// TIA Portal V18 export
FUNCTION_BLOCK "Control_Buttons_Manipulate"   // FB24, LAD
{ S7_Optimized_Access := 'TRUE' }
VERSION : 0.1
// Simple control block to activate printhead motion in X and Y direction
// stored: AutoNumber true, IsIECCheckEnabled false, IsRetainMemResEnabled false, MemoryReserve 100, SetENOAutomatically false, UDAEnableTagReadback false
   VAR_INPUT
      JogInZ1pos : Bool;
      JogInZ1neg : Bool;
      JogInZ2pos : Bool;
      JogInZ2neg : Bool;
      InXhome : Bool;
      InYhome : Bool;
      InZ1home : Bool;
      InZ2home : Bool;
      MovePermission : Bool;
      ReadyDevices : Bool;
   END_VAR
   VAR_OUTPUT
      JogOutXpos : Bool;
      JogOutXneg : Bool;
      JogOutYpos : Bool;
      JogOutYneg : Bool;
      JogOutZ1pos : Bool;
      JogOutZ1neg : Bool;
      JogOutZ2pos : Bool;
      JogOutZ2neg : Bool;
      XHoming : Bool;
      YHoming : Bool;
      Z1Homing : Bool;
      Z2Homing : Bool;
      StartMachine : Bool;
   END_VAR
   VAR
      ButtonsReadyToRead : Bool;
      XYmoveout : Bool;
   END_VAR
BEGIN

REGION Network 1: Start Machine
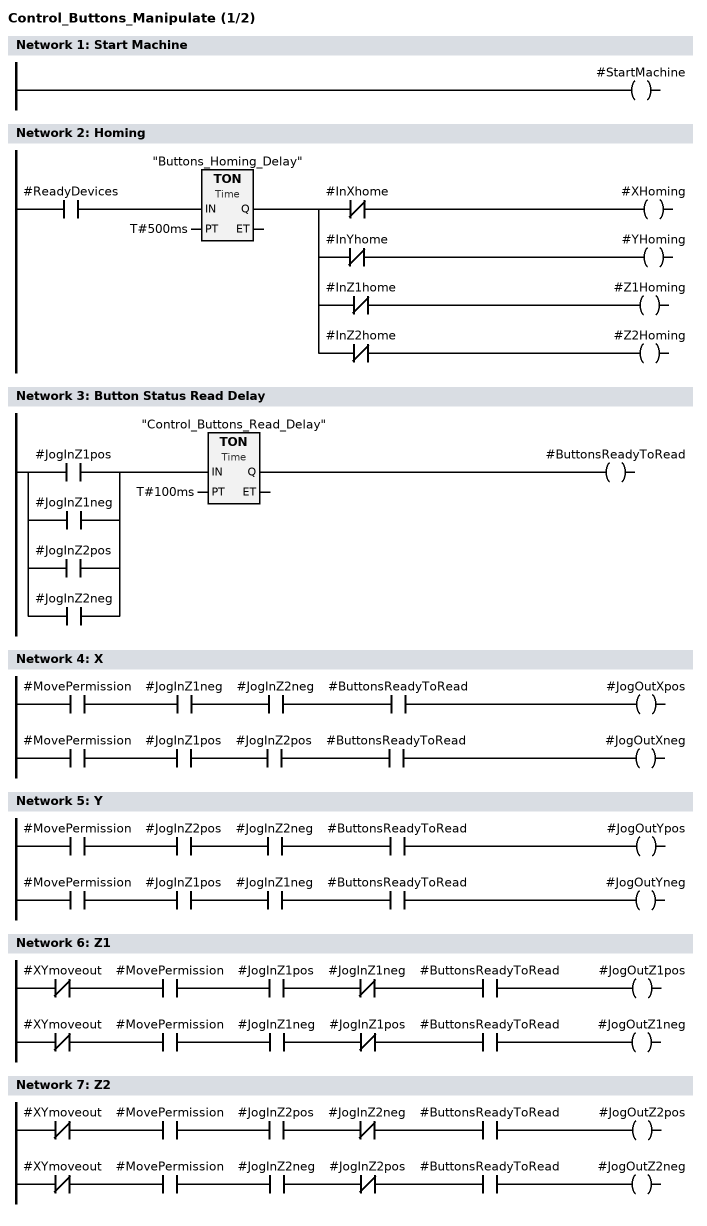
   RUNG wire#powerrail
      Coil( #StartMachine )
   END_RUNG
   // the same network as SCL:
   #StartMachine := TRUE;
END_REGION

REGION Network 2: Homing
   RUNG wire#powerrail
      Contact( #ReadyDevices )
      { S7_Templates := "time_type := Time" } "Buttons_Homing_Delay".TON(pt := T#500ms, et =>)
      wire#w1
      I_Contact( #InXhome )
      Coil( #XHoming )
   END_RUNG
   RUNG wire#w1
      I_Contact( #InYhome )
      Coil( #YHoming )
   END_RUNG
   RUNG wire#w1
      I_Contact( #InZ1home )
      Coil( #Z1Homing )
   END_RUNG
   RUNG wire#w1
      I_Contact( #InZ2home )
      Coil( #Z2Homing )
   END_RUNG
   // the same network as SCL:
   "Buttons_Homing_Delay".TON(IN := #ReadyDevices, PT := T#500ms);
   #XHoming := "Buttons_Homing_Delay".Q AND NOT #InXhome;
   #YHoming := "Buttons_Homing_Delay".Q AND NOT #InYhome;
   #Z1Homing := "Buttons_Homing_Delay".Q AND NOT #InZ1home;
   #Z2Homing := "Buttons_Homing_Delay".Q AND NOT #InZ2home;
END_REGION

REGION Network 3: Button Status Read Delay
   RUNG wire#powerrail
      Contact( #JogInZ1pos )
      wire#w1
      { S7_Templates := "time_type := Time" } "Control_Buttons_Read_Delay".TON(pt := T#100ms, et =>)
      Coil( #ButtonsReadyToRead )
   END_RUNG
   RUNG wire#powerrail
      Contact( #JogInZ1neg )
   END_RUNG wire#w1
   RUNG wire#powerrail
      Contact( #JogInZ2pos )
   END_RUNG wire#w1
   RUNG wire#powerrail
      Contact( #JogInZ2neg )
   END_RUNG wire#w1
   // the same network as SCL:
   "Control_Buttons_Read_Delay".TON(IN := #JogInZ1pos OR #JogInZ1neg OR #JogInZ2pos OR #JogInZ2neg,
                           PT := T#100ms);
   #ButtonsReadyToRead := "Control_Buttons_Read_Delay".Q;
END_REGION

REGION Network 4: X
   RUNG wire#powerrail
      Contact( #MovePermission )
      Contact( #JogInZ1neg )
      Contact( #JogInZ2neg )
      Contact( #ButtonsReadyToRead )
      Coil( #JogOutXpos )
   END_RUNG
   RUNG wire#powerrail
      Contact( #MovePermission )
      Contact( #JogInZ1pos )
      Contact( #JogInZ2pos )
      Contact( #ButtonsReadyToRead )
      Coil( #JogOutXneg )
   END_RUNG
   // the same network as SCL:
   #JogOutXpos := #MovePermission AND #JogInZ1neg AND #JogInZ2neg AND #ButtonsReadyToRead;
   #JogOutXneg := #MovePermission AND #JogInZ1pos AND #JogInZ2pos AND #ButtonsReadyToRead;
END_REGION

REGION Network 5: Y
   RUNG wire#powerrail
      Contact( #MovePermission )
      Contact( #JogInZ2pos )
      Contact( #JogInZ2neg )
      Contact( #ButtonsReadyToRead )
      Coil( #JogOutYpos )
   END_RUNG
   RUNG wire#powerrail
      Contact( #MovePermission )
      Contact( #JogInZ1pos )
      Contact( #JogInZ1neg )
      Contact( #ButtonsReadyToRead )
      Coil( #JogOutYneg )
   END_RUNG
   // the same network as SCL:
   #JogOutYpos := #MovePermission AND #JogInZ2pos AND #JogInZ2neg AND #ButtonsReadyToRead;
   #JogOutYneg := #MovePermission AND #JogInZ1pos AND #JogInZ1neg AND #ButtonsReadyToRead;
END_REGION

REGION Network 6: Z1
   RUNG wire#powerrail
      I_Contact( #XYmoveout )
      Contact( #MovePermission )
      Contact( #JogInZ1pos )
      I_Contact( #JogInZ1neg )
      Contact( #ButtonsReadyToRead )
      Coil( #JogOutZ1pos )
   END_RUNG
   RUNG wire#powerrail
      I_Contact( #XYmoveout )
      Contact( #MovePermission )
      Contact( #JogInZ1neg )
      I_Contact( #JogInZ1pos )
      Contact( #ButtonsReadyToRead )
      Coil( #JogOutZ1neg )
   END_RUNG
   // the same network as SCL:
   #JogOutZ1pos := NOT #XYmoveout AND #MovePermission AND #JogInZ1pos AND NOT #JogInZ1neg AND #ButtonsReadyToRead;
   #JogOutZ1neg := NOT #XYmoveout AND #MovePermission AND #JogInZ1neg AND NOT #JogInZ1pos AND #ButtonsReadyToRead;
END_REGION

REGION Network 7: Z2
   RUNG wire#powerrail
      I_Contact( #XYmoveout )
      Contact( #MovePermission )
      Contact( #JogInZ2pos )
      I_Contact( #JogInZ2neg )
      Contact( #ButtonsReadyToRead )
      Coil( #JogOutZ2pos )
   END_RUNG
   RUNG wire#powerrail
      I_Contact( #XYmoveout )
      Contact( #MovePermission )
      Contact( #JogInZ2neg )
      I_Contact( #JogInZ2pos )
      Contact( #ButtonsReadyToRead )
      Coil( #JogOutZ2neg )
   END_RUNG
   // the same network as SCL:
   #JogOutZ2pos := NOT #XYmoveout AND #MovePermission AND #JogInZ2pos AND NOT #JogInZ2neg AND #ButtonsReadyToRead;
   #JogOutZ2neg := NOT #XYmoveout AND #MovePermission AND #JogInZ2neg AND NOT #JogInZ2pos AND #ButtonsReadyToRead;
END_REGION

REGION Network 8: Status
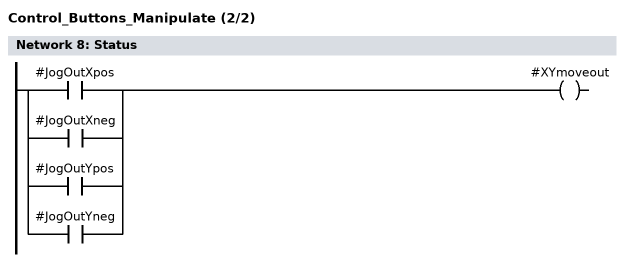
   RUNG wire#powerrail
      Contact( #JogOutXpos )
      wire#w1
      Coil( #XYmoveout )
   END_RUNG
   RUNG wire#powerrail
      Contact( #JogOutXneg )
   END_RUNG wire#w1
   RUNG wire#powerrail
      Contact( #JogOutYpos )
   END_RUNG wire#w1
   RUNG wire#powerrail
      Contact( #JogOutYneg )
   END_RUNG wire#w1
   // the same network as SCL:
   #XYmoveout := #JogOutXpos OR #JogOutXneg OR #JogOutYpos OR #JogOutYneg;
END_REGION
END_FUNCTION_BLOCK
